// TIA Portal V21 export
FUNCTION "Main sequenze" : Void   // FC91, LAD
{ S7_Optimized_Access := 'TRUE' }
// stored: SetENOAutomatically false
   VAR_TEMP
      Indice_SequenzaAttuale : Int;
      Hmi_SequenzaAttuale : Int;
      Hmi_PassoAttuale : Int;
   END_VAR
BEGIN
END_FUNCTION
